(* IEC 61131-3 sources: Word/plc-course/09-math-and-data-handling/labs/solutions, 3 files *)

(* ---- 09-1-scaling-function.st ---- *)
(* Lab 09-1: A general scaling function, F_Scale.
   Module 09 (Maths, comparison, data movement and bit manipulation).
   REFERENCE SOLUTION - try the lab yourself first.

   One function does every straight-line conversion in the program:
     raw counts -> metres     (level, not clamped, so over-range stays visible)
     raw counts -> percent    (bar graph, clamped)
     hertz      -> raw counts (drive speed reference, clamped)
     percent    -> raw counts (reverse-acting valve: 0 % open = 20 mA)

   Raw-count convention (as in Module 14): 0..27648 = 4..20 mA. *)

FUNCTION F_Scale : REAL
  VAR_INPUT
    In     : REAL;   (* the value to convert *)
    InMin  : REAL;   (* input value that corresponds to OutMin *)
    InMax  : REAL;   (* input value that corresponds to OutMax *)
    OutMin : REAL;   (* result when In = InMin *)
    OutMax : REAL;   (* result when In = InMax *)
    Clamp  : BOOL;   (* TRUE: keep the result inside the output range *)
  END_VAR
  VAR
    InSpan : REAL;
    Result : REAL;
  END_VAR

  InSpan := InMax - InMin;

  (* Divide-by-zero protection. A span of exactly 0.0 is the one case that
     makes the division below return infinity or NaN, so this is one of the
     few places where "=" on a REAL is the right test. A bad configuration
     gives the bottom of the output range: a defined, visible value. *)
  IF InSpan = 0.0 THEN
    Result := OutMin;
  ELSE
    (* y = (x - x0) * (y1 - y0) / (x1 - x0) + y0, all in REAL *)
    Result := (In - InMin) * (OutMax - OutMin) / InSpan + OutMin;
  END_IF;

  (* Clamp to the output range. OutMin may be larger than OutMax (a
     reverse-acting output), so find the lower and upper bounds first:
     LIMIT(MN, IN, MX) needs MN <= MX. *)
  IF Clamp THEN
    Result := LIMIT(MIN(OutMin, OutMax), Result, MAX(OutMin, OutMax));
  END_IF;

  F_Scale := Result;
END_FUNCTION

PROGRAM ScalingDemo
  VAR (* I/O *)
    LevelRaw AT %IW0 : INT;   (* LT-101 tank level, raw counts from the analog input card *)
    SpeedAO  AT %QW0 : INT;   (* SC-103 drive speed reference, raw counts: 0..27648 = 4..20 mA *)
    ValveAO  AT %QW1 : INT;   (* FV-102 valve demand, raw counts: 0 = 4 mA = fully OPEN *)
  END_VAR
  VAR (* settings: configuration of the card, the transmitter and the drive *)
    RawAt4mA   : REAL := 0.0;      (* raw count the card gives at 4 mA *)
    RawAt20mA  : REAL := 27648.0;  (* raw count the card gives at 20 mA *)
    DriveMinHz : REAL := 0.0;      (* drive speed at 4 mA (drive parameter) *)
    DriveMaxHz : REAL := 50.0;     (* drive speed at 20 mA (drive parameter) *)
  END_VAR
  VAR (* HMI values *)
    Level_m      : REAL;           (* LT-101 level in metres, NOT clamped *)
    LevelPct     : REAL;           (* LT-101 level in % of range, clamped 0..100 for the bar graph *)
    SpeedRef_Hz  : REAL;           (* speed setpoint entered on the HMI *)
    ValveCmd_Pct : REAL;           (* valve opening demand: 0 = closed, 100 = fully open *)
  END_VAR
  VAR CONSTANT
    LEVEL_MIN_M : REAL := 0.5;     (* LT-101 range: 0.5 m at 4 mA (the tapping is 0.5 m above the floor) ... *)
    LEVEL_MAX_M : REAL := 4.5;     (* ... 4.5 m at 20 mA *)
    AO_RAW_4MA  : REAL := 0.0;     (* analog output raw count for 4 mA *)
    AO_RAW_20MA : REAL := 27648.0; (* analog output raw count for 20 mA *)
  END_VAR

  (* Level for the operator and for alarms: not clamped, so a reading of
     4.7 m or 0.3 m shows that the transmitter or loop needs attention
     (Module 14: check the signal before you clamp it). *)
  Level_m := F_Scale(In := INT_TO_REAL(LevelRaw),
                     InMin := RawAt4mA, InMax := RawAt20mA,
                     OutMin := LEVEL_MIN_M, OutMax := LEVEL_MAX_M,
                     Clamp := FALSE);

  (* Bar graph: clamped so it never shows -3 % or 106 %. *)
  LevelPct := F_Scale(In := INT_TO_REAL(LevelRaw),
                      InMin := RawAt4mA, InMax := RawAt20mA,
                      OutMin := 0.0, OutMax := 100.0,
                      Clamp := TRUE);

  (* Drive speed reference: clamped, so a mistyped 500 Hz can never send more
     than 20 mA. The clamp is applied to the REAL before REAL_TO_INT, which
     also keeps the conversion inside the INT range. *)
  SpeedAO := REAL_TO_INT(F_Scale(In := SpeedRef_Hz,
                                 InMin := DriveMinHz, InMax := DriveMaxHz,
                                 OutMin := AO_RAW_4MA, OutMax := AO_RAW_20MA,
                                 Clamp := TRUE));

  (* Reverse-acting valve: 0 % open needs 20 mA and 100 % open needs 4 mA,
     so the output range is simply given "upside down". *)
  ValveAO := REAL_TO_INT(F_Scale(In := ValveCmd_Pct,
                                 InMin := 0.0, InMax := 100.0,
                                 OutMin := AO_RAW_20MA, OutMax := AO_RAW_4MA,
                                 Clamp := TRUE));
END_PROGRAM

CONFIGURATION Config0
  RESOURCE Res0 ON PLC
    TASK MainTask(INTERVAL := T#10ms, PRIORITY := 0);
    PROGRAM Inst0 WITH MainTask : ScalingDemo;
  END_RESOURCE
END_CONFIGURATION

(* ---- 09-2-reject-tracking.st ---- *)
(* Lab 09-2: Conveyor reject tracking with a bit shift register.
   Module 09 (Maths, comparison, data movement and bit manipulation).
   REFERENCE SOLUTION - try the lab yourself first.

   Parts travel on a conveyor one pitch apart. A camera at position 0 checks
   each part; the reject pusher is RejectPos pitches further down the belt.
   Each bit of TrackWord stands for one position on the belt:

      bit:      15  ...  6   5   4   3   2   1   0
      position: 15  ...  6   5   4   3   2   1   0 (camera)
                              ^ reject gate (RejectPos = 5)

   A bad result sets bit 0. Every pitch of belt movement (one rising edge of
   EncoderPulse) shifts the word one place left, so the "bad" bit travels
   down the belt with its part. The gate fires while the bit at RejectPos
   is set. *)

PROGRAM RejectTracking
  VAR (* I/O *)
    EncoderPulse AT %IX0.0 : BOOL;  (* one pulse per pitch, from a prox on the drive sprocket *)
    InspectFail  AT %IX0.1 : BOOL;  (* camera at position 0: TRUE = the part in front of it failed *)
    ResetPB      AT %IX0.2 : BOOL;  (* clear the tracking after the belt has been emptied by hand *)
    RejectGate   AT %QX0.0 : BOOL;  (* reject pusher at position RejectPos *)
  END_VAR
  VAR (* settings and HMI values *)
    RejectPos   : INT := 5;         (* pitches from the camera to the reject gate, 1..15 *)
    TrackWord   : WORD;             (* bit n TRUE = the part n pitches past the camera is bad *)
    RejectCount : DINT;             (* bad parts that have reached the reject gate *)
  END_VAR
  VAR (* internal *)
    PulseEdge : R_TRIG;             (* the belt has moved one pitch *)
    GatePos   : INT;                (* RejectPos limited to the bits that exist *)
    GateMask  : WORD;               (* a single 1 in bit GatePos *)
  END_VAR

  (* 1. Which bit is the gate? LIMIT keeps a bad setting inside the word:
        SHL by 16 or more would give a mask of 0, and the gate would never
        fire again. *)
  GatePos := LIMIT(1, RejectPos, 15);
  GateMask := SHL(WORD#16#0001, GatePos);

  (* 2. Mark: a fail from the camera sets bit 0, the part at the camera.
        OR sets that one bit and leaves the other fifteen alone. *)
  IF InspectFail THEN
    TrackWord := TrackWord OR WORD#16#0001;
  END_IF;

  (* 3. Shift once per pitch, on the rising edge only: a pulse that stays on
        while the belt is stopped must not shift the word every scan.
        SHL (not ROL) lets the bit from position 15 fall off the end, and
        brings a 0 (not yet inspected, so not bad) into bit 0.
        Marking comes first, so a camera result that arrives in the same scan
        as the pulse stays with the part it was taken of. *)
  PulseEdge(CLK := EncoderPulse);
  IF PulseEdge.Q THEN
    TrackWord := SHL(TrackWord, 1);
    (* Count here, once per shift, and not on the gate's rising edge: two
       bad parts in a row keep the gate on, but they are two rejects. *)
    IF (TrackWord AND GateMask) <> WORD#16#0000 THEN
      RejectCount := RejectCount + 1;
    END_IF;
  END_IF;

  (* 4. Reset clears the tracking only. The count is production data. *)
  IF ResetPB THEN
    TrackWord := WORD#16#0000;
  END_IF;

  (* 5. The gate follows the bit at its position. *)
  RejectGate := (TrackWord AND GateMask) <> WORD#16#0000;
END_PROGRAM

CONFIGURATION Config0
  RESOURCE Res0 ON PLC
    TASK MainTask(INTERVAL := T#10ms, PRIORITY := 0);
    PROGRAM Inst0 WITH MainTask : RejectTracking;
  END_RESOURCE
END_CONFIGURATION

(* ---- 09-3-flow-totaliser.st ---- *)
(* Lab 09-3: Flow totaliser.
   Module 09 (Maths, comparison, data movement and bit manipulation).
   REFERENCE SOLUTION - try the lab yourself first.

   A totaliser integrates a rate over time. Every scan:

       increment [m3] = flow [m3/h] x scan time [h]

   With a 10 ms task the increment is tiny (50 m3/h adds 0.000139 m3 per
   scan), and that is exactly what a REAL cannot add to a large number:
   a REAL keeps about 7 significant digits, so near 20000 m3 the gap between
   neighbouring REAL values is about 0.002 m3 and every increment is rounded
   away. This program keeps two totals side by side:
     Total_m3      in LREAL (about 16 digits): correct
     TotalReal_m3  in REAL, the naive way: shown only so you can watch it fail *)

PROGRAM FlowTotaliser
  VAR (* I/O *)
    ResetPB  AT %IX0.0 : BOOL;       (* reset the totaliser to zero (NO key switch) *)
    PresetPB AT %IX0.1 : BOOL;       (* load PresetValue_m3 into the totaliser (NO) *)
  END_VAR
  VAR (* process value and settings *)
    FlowRate       : REAL;           (* FT-201 flow in m3/h, already scaled (Module 14) *)
    PresetValue_m3 : DINT;           (* whole m3 to load, e.g. the reading of the meter being replaced *)
    TaskCycle      : TIME := T#10ms; (* the task interval: must match the TASK INTERVAL below *)
  END_VAR
  VAR RETAIN (* on a real PLC the totals must survive a power cut *)
    Total_m3     : LREAL;            (* the accurate total, m3 *)
    TotalReal_m3 : REAL;             (* the naive REAL total, m3: for comparison only *)
  END_VAR
  VAR (* outputs for SCADA and the HMI *)
    TotalWhole_m3 : DINT;            (* whole cubic metres of Total_m3, like a meter's counter *)
  END_VAR
  VAR (* internal *)
    Dt_h     : LREAL;                (* scan time in hours *)
    Flow     : REAL;                 (* the flow that is totalised: never negative *)
  END_VAR

  (* 1. Scan time in hours. TIME_TO_LREAL returns seconds in MATIEC but
        milliseconds in CODESYS; the ratio of two conversions is the same on
        every platform, so this line is portable. *)
  Dt_h := TIME_TO_LREAL(TaskCycle) / TIME_TO_LREAL(T#1h);

  (* 2. Only forward flow is totalised. A small negative reading around zero
        flow is noise, not flow going backwards. Writing the test as
        "FlowRate > 0.0" also means a NaN flow (every comparison with NaN is
        FALSE) counts as zero instead of turning the total into NaN for ever. *)
  IF FlowRate > 0.0 THEN
    Flow := FlowRate;
  ELSE
    Flow := 0.0;
  END_IF;

  (* 3. Reset wins over preset; while either is held, nothing is added. *)
  IF ResetPB THEN
    Total_m3 := 0.0;
    TotalReal_m3 := 0.0;
  ELSIF PresetPB THEN
    Total_m3 := DINT_TO_LREAL(PresetValue_m3);
    TotalReal_m3 := DINT_TO_REAL(PresetValue_m3);
  ELSE
    (* The accurate total: the whole calculation in LREAL. *)
    Total_m3 := Total_m3 + REAL_TO_LREAL(Flow) * Dt_h;
    (* The naive total: the same sum in REAL. It is fine while the total is
       small, then loses increments, then stops counting altogether. *)
    TotalReal_m3 := TotalReal_m3 + Flow * LREAL_TO_REAL(Dt_h);
  END_IF;

  (* 4. Whole cubic metres, cut off (not rounded) like a mechanical counter:
        7.9 m3 shows 7 until the eighth cubic metre is complete. *)
  TotalWhole_m3 := TRUNC(Total_m3);
END_PROGRAM

CONFIGURATION Config0
  RESOURCE Res0 ON PLC
    TASK MainTask(INTERVAL := T#10ms, PRIORITY := 0);
    PROGRAM Inst0 WITH MainTask : FlowTotaliser;
  END_RESOURCE
END_CONFIGURATION
